Universal Robots PolyScope program: 20250523mode2.urp

Program 20250523mode2 (installation=20240827 directory=/programs/collection createdIn=5.15.1 lastSavedIn=5.15.1 robotSerialNumber=20245500285)
Calibrated DH parameters: a=[0.000097, -0.210459, -0.026602, 0.000137, 0.000078, 0]; d=[0.162601, 254.180657, -54.076236, -199.970743, 0.099615, 0.099684]; alpha=[1.569796, -0.001455, 0.001957, 1.570525, -1.571561, 0]; deltaTheta=[0, -1.053331, 8.839472, -1.50296, 0.000002, 0]
InitVariablesNode
Robot Program (runOnlyOnce=false)
  mode := 0
  '0-空闲/1-基础验证/2-中心点Z/3-全点Z'
  step_x := 0.004
  step_y := 0.004
  step_z := 0.0002
  step_tcp := 0.0001
  var_x := [0,-1,1,-1,1,0]
  var_y := [0,-1,1,1,-1,0]
  '一维路点(0,0)(-1,1)(1,1)(-1,-1)(1,-1)'
  '默认一维路点(0,0)'
  Popup Message (haltProgram=false inputType=Variable) variable=mode
  MoveJ speed 60 deg/s, acceleration 80 deg/s^2 (useActiveTCP=true) feature=Base
    Waypoint 路点_1: TCP in base x=804.825 y=122.722 z=261.377 mm, rx=1.21 ry=1.2107 rz=1.2121 rad; joints [178.75, -48.538, 102.99, -234.413, -88.607, 180.11] deg; TCP offset x=-0.17 y=0 z=192.95 mm, rx=0 ry=0 rz=0 rad
    '过渡点'
    Waypoint tcp: TCP in base x=804.822 y=122.747 z=254.96 mm, rx=1.2099 ry=1.2106 rz=1.2122 rad; joints [178.646, -47.791, 103.049, -235.262, -88.649, 180.008] deg
    '受力0，距离0'
  If mode==0
    Popup Message (haltProgram=false message=空闲模式 inputType=Text)
  ElseIf mode==1
    Popup Message (haltProgram=false message=基础TCP位置验证 inputType=Text)
    step := 0
    Loop Counting (count=20) loopVariable(name=循环_1)
      step := step+1
      tcptcp := pose_add(tcp, p[0,0,-step_tcp*step,0,0,0])
      MoveJ speed 60 deg/s, acceleration 80 deg/s^2 (useActiveTCP=true) feature=Base
        Popup Message (haltProgram=false inputType=Variable) variable(name=tcptcp)
        Waypoint Variable (Variable): variable(name=tcptcp)
    Popup Message (haltProgram=false message=基础TCP位置验证 inputType=Text)
  ElseIf mode==2
    Popup Message (haltProgram=false message=中心点Z方向测试 inputType=Text)
    step := 0
    Loop Counting (count=25) loopVariable(name=循环_2)
      step := step+1
      tcptcp := pose_add(tcp, p[0,0,-step*step_z,0,0,0])
      MoveJ speed 60 deg/s, acceleration 80 deg/s^2 (useActiveTCP=true) feature=Base
        Popup Message (haltProgram=false inputType=Variable) variable=tcptcp
        Waypoint Variable (Variable): variable=tcptcp
    Popup Message (haltProgram=false message=中心点Z方向测试 inputType=Text)
  ElseIf mode==3
    Popup Message (haltProgram=false message=全点Z测试 inputType=Text)
    xy := 0
    Loop Counting (count=5) loopVariable(name=循环_4)
      MoveJ speed 60 deg/s, acceleration 80 deg/s^2 (useActiveTCP=true) feature=Base
        Waypoint 路点_1: TCP in base x=804.825 y=122.722 z=261.377 mm, rx=1.21 ry=1.2107 rz=1.2121 rad; joints [178.75, -48.538, 102.99, -234.413, -88.607, 180.11] deg
      xy := xy+1
      step := 0
      Loop Counting (count=25) loopVariable(name=循环_5)
        step := step+1
        tcptcp := pose_add(tcp, p[step_x*var_x[xy],step_y*var_y[xy],-step*step_z,0,0,0])
        MoveJ speed 60 deg/s, acceleration 80 deg/s^2 (useActiveTCP=true) feature=Base
          Popup Message (haltProgram=false inputType=Variable) variable=tcptcp
          Waypoint Variable (Variable): variable=tcptcp
    Popup Message (haltProgram=false message=全点Z测试 inputType=Text)
